FUNCTION_BLOCK TCPIP_Base IMPLEMENTS ITF_TcpIpBase
VAR_INPUT
END_VAR
VAR_OUTPUT
END_VAR
VAR
	connectToServer : SocketConnectTask;
	closeConectionToServer : SocketCloseTask;
	getReceivedDataFromServer : SocketRecieveTask;
	sendDataToServer : SocketSendTask;
	iState : INT;
	_connect: BOOL;
	_remoteIP : T_IPv4Addr;
	_remotePort : UDINT;
	_remoteHandle : Tc2_TcpIp.T_HSOCKET;
	clearRecieve: BOOL;
	_disconnect: BOOL;
	_connected: BOOL;
END_VAR

CASE iState OF
	0: 
		IF _connect THEN
			_connect := false;
			iState := 10;
		END_IF
		
	10:
		IF connectToServer.Execute(RemoteIPAddress := _remoteIP, 
									RemotePortNumber := _remotePort) THEN
			iState := 20;
		END_IF
		
	20:
		_remoteHandle := connectToServer.RemoteSocket;
		getReceivedDataFromServer.RemoteSocket := _remoteHandle;
		IF connectToServer.Done AND _remoteHandle.handle <> 0 THEN
			iState := 30;
			_connected := TRUE;
		END_IF
	
	30:
		IF getReceivedDataFromServer.Execute() THEN
			iState := 40;
		END_IF
		
	40:
		IF getReceivedDataFromServer.Done THEN
			IF _disconnect THEN
				_disconnect := FALSE;
				iState := 50;
			ELSE
				iState := 30;
			END_IF
			
		END_IF
	
	50:
		IF closeConectionToServer.Execute(remoteSocket := _remoteHandle) THEN
			iState := 60;
		END_IF
		
	60:
		IF closeConectionToServer.Done THEN
			iState := 0;
			_connected := FALSE;
		END_IF
		
			
END_CASE

connectToServer();
closeConectionToServer();
getReceivedDataFromServer();
sendDataToServer();

METHOD ConnectToRobot : BOOL
VAR_INPUT
END_VAR
ConnectToRobot := _connect := true;
END_METHOD

METHOD DisconnectFromRobot : BOOL
VAR_INPUT
END_VAR
DisconnectFromRobot := _disconnect := true;
END_METHOD

METHOD PUBLIC GetData : ARRAY[0..1439] OF byte
VAR_INPUT
END_VAR
GetData := getReceivedDataFromServer.rxBuffer;
END_METHOD

METHOD PUBLIC IsConnected : BOOL
VAR_INPUT
END_VAR
IsConnected := _connected;
END_METHOD

PROPERTY PUBLIC RemoteServerIP : T_IPv4Addr
GET
RemoteServerIP := _remoteIP;
END_GET
SET
_remoteIP := RemoteServerIP;
END_SET
END_PROPERTY

PROPERTY PUBLIC RemoteServerPort : udint
GET
RemoteServerPort := _remotePort;
END_GET
SET
_remotePort := RemoteServerPort;
END_SET
END_PROPERTY

END_FUNCTION_BLOCK

(* stored: Version 1.1.0.1, ProductVersion 3.1.4024.12
   POU TCPIP_Base: Id {65da1431-803c-4746-bb7f-22bf27a0e177}, SpecialFunc None
   Method ConnectToRobot: Id {0e802047-5a08-436c-8d42-86478532b47e}
   Method DisconnectFromRobot: Id {6491f002-ea1e-4b9f-8dee-8bcb7cc1dea4}
   Method GetData: Id {8cdab55b-3cfc-400c-b81e-4f087af29019}
   Method IsConnected: Id {d4afbbff-19b5-479d-8d61-a567ab11d390}
   Property RemoteServerIP: Id {c712af6f-cb00-48f5-a7f0-31ace650ed71}
   Get Get: Id {2869d66b-9724-44d0-b781-254c975a5157}
   Set Set: Id {afc45aa6-07cd-4ce8-bee8-975fe3a8c50d}
   Property RemoteServerPort: Id {2499f905-4fde-4178-984c-0ea485973f73}
   Get Get: Id {20744aaa-48ec-4835-a6ac-d9a791159548}
   Set Set: Id {a7ef5c8d-1f8f-4dab-82bc-c617e0cd9f5c} *)
